// TIA Portal project "FLASOR YAPMA" (V18)
// belirli bir sure yanan belirli bir sure de sonen lamba dusunebilirz plc cikisina baglanan.

(* hardware
DEVICE "S7-1200 station_1"  S7-1200 Station
   slot 0: "Rack_0"  S7-1200 Rack  Rack  V1.0
   slot 1: "PLC_1"  CPU 1212C DC/DC/DC  6ES7 212-1AE40-0XB0  V4.6
*)

// ===== PLC "PLC_1"  CPU 1212C DC/DC/DC =====

VAR_GLOBAL   // PLC tag table "Default tag table"
   "START BUT" AT %I0.0 : Bool;
   "STOP BUT" AT %I0.1 : Bool;
   "SISTEM MEM" AT %M10.0 : Bool;
   "FLASOR" AT %Q0.0 : Bool;
END_VAR

// folder: System blocks/Program resources

DATA_BLOCK "TIMER 1"   // DB1
{ S7_Optimized_Access := 'TRUE' }
AUTHOR : Simatic
FAMILY : IEC
NAME : IEC_TMR
VERSION : 1.0
// stored: InstanceOfName IEC_TIMER
"IEC_TIMER"
BEGIN
END_DATA_BLOCK

DATA_BLOCK "TIMER 2"   // DB2
{ S7_Optimized_Access := 'TRUE' }
AUTHOR : Simatic
FAMILY : IEC
NAME : IEC_TMR
VERSION : 1.0
// stored: InstanceOfName IEC_TIMER
"IEC_TIMER"
BEGIN
END_DATA_BLOCK

// folder: (top level)

ORGANIZATION_BLOCK "Main"   // OB1, LAD, ProgramCycle
TITLE = "Main Program Sweep (Cycle)"
{ S7_Optimized_Access := 'TRUE' }
VERSION : 0.1
   VAR_INPUT
      Initial_Call : Bool;   // Initial call of this OB
      Remanence : Bool;   // =True, if remanent data are available
   END_VAR
BEGIN

REGION Network 1: SISTEM HAZIR MEMEORY
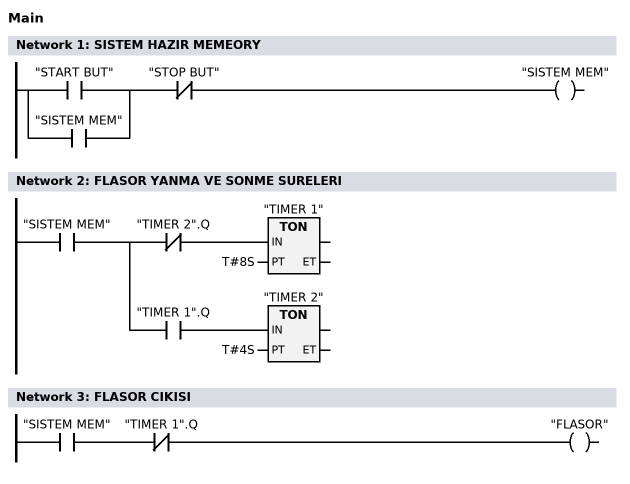
   RUNG wire#powerrail
      Contact( "START BUT" )
      wire#w1
      I_Contact( "STOP BUT" )
      Coil( "SISTEM MEM" )
   END_RUNG
   RUNG wire#powerrail
      Contact( "SISTEM MEM" )
   END_RUNG wire#w1
   // the same network as SCL:
   "SISTEM MEM" := ("START BUT" OR "SISTEM MEM") AND NOT "STOP BUT";
END_REGION

REGION Network 2: FLASOR YANMA VE SONME SURELERI
   "TIMER 1".TON(IN := "SISTEM MEM" AND NOT "TIMER 2".Q, PT := T#8S);
   "TIMER 2".TON(IN := "SISTEM MEM" AND "TIMER 1".Q, PT := T#4S);
END_REGION

REGION Network 3: FLASOR CIKISI
   RUNG wire#powerrail
      Contact( "SISTEM MEM" )
      I_Contact( "TIMER 1".Q )
      Coil( "FLASOR" )
   END_RUNG
   // the same network as SCL:
   "FLASOR" := "SISTEM MEM" AND NOT "TIMER 1".Q;
END_REGION
END_ORGANIZATION_BLOCK